TEXTLIST MoveType
  0 = 'Circular'
  1 = 'Direct'
  2 = 'Linear'
   = ''
END_TEXTLIST

(* stored: Version 1.1.0.1
   TextList MoveType: Id {9d428ec6-1ee8-423e-96f6-af8930972a16} *)
